// TIA Portal V18 export
TYPE "UDT_Vitotronic100_Settings"
// stored: IsFailsafeCompliant false
   STRUCT
      "Set boiler water temperature" : Array[0..2] of Real;
      "Operating mode system_boiler" : Array[0..2] of Int;
   END_STRUCT;
END_TYPE
